SUBAPPLICATION Uebung_003b3_AX (* Funk 16 Tasten auf DataPanel 16 *)
  (* Standard: 61499-2; Description: Copyright (c) 2023 Meisterschulen am Ostbahnhof This program and the accompanying materials are made available under the terms of the Eclipse Public License 2.0 which is available at https://www.eclipse.org/legal/epl-2.0/ SPDX-License-Identifier: EPL-2.0 *)
  (* Version 1.0, 2023-10-23, Franz Höpfinger, Meisterschulen am Ostbahnhof *)
  PACKAGE Uebungen;
  IMPORT DataPanel::io::MI::DQ::DataPanel_MI_DO::DigitalOutput_1A;
  IMPORT DataPanel::io::MI::DQ::DataPanel_MI_DO::DigitalOutput_1B;
  IMPORT DataPanel::io::MI::DQ::DataPanel_MI_DO::DigitalOutput_2A;
  IMPORT DataPanel::io::MI::DQ::DataPanel_MI_DO::DigitalOutput_2B;
  IMPORT DataPanel::io::MI::DQ::DataPanel_MI_DO::DigitalOutput_3A;
  IMPORT DataPanel::io::MI::DQ::DataPanel_MI_DO::DigitalOutput_3B;
  IMPORT DataPanel::io::MI::DQ::DataPanel_MI_DO::DigitalOutput_4A;
  IMPORT DataPanel::io::MI::DQ::DataPanel_MI_DO::DigitalOutput_4B;
  IMPORT DataPanel::io::MI::DQ::DataPanel_MI_DO::DigitalOutput_5A;
  IMPORT DataPanel::io::MI::DQ::DataPanel_MI_DO::DigitalOutput_5B;
  IMPORT DataPanel::io::MI::DQ::DataPanel_MI_DO::DigitalOutput_6A;
  IMPORT DataPanel::io::MI::DQ::DataPanel_MI_DO::DigitalOutput_6B;
  IMPORT DataPanel::io::MI::DQ::DataPanel_MI_DO::DigitalOutput_7A;
  IMPORT DataPanel::io::MI::DQ::DataPanel_MI_DO::DigitalOutput_7B;
  IMPORT DataPanel::io::MI::DQ::DataPanel_MI_DO::DigitalOutput_8A;
  IMPORT DataPanel::io::MI::const::MI::MI_00;
  IMPORT Funk::io::DI::Funk_DI::DigitalInput_Key_01;
  IMPORT Funk::io::DI::Funk_DI::DigitalInput_Key_02;
  IMPORT Funk::io::DI::Funk_DI::DigitalInput_Key_03;
  IMPORT Funk::io::DI::Funk_DI::DigitalInput_Key_04;
  IMPORT Funk::io::DI::Funk_DI::DigitalInput_Key_05;
  IMPORT Funk::io::DI::Funk_DI::DigitalInput_Key_06;
  IMPORT Funk::io::DI::Funk_DI::DigitalInput_Key_07;
  IMPORT Funk::io::DI::Funk_DI::DigitalInput_Key_08;
  IMPORT Funk::io::DI::Funk_DI::DigitalInput_Key_09;
  IMPORT Funk::io::DI::Funk_DI::DigitalInput_Key_10;
  IMPORT Funk::io::DI::Funk_DI::DigitalInput_Key_11;
  IMPORT Funk::io::DI::Funk_DI::DigitalInput_Key_12;
  IMPORT Funk::io::DI::Funk_DI::DigitalInput_Key_13;
  IMPORT Funk::io::DI::Funk_DI::DigitalInput_Key_14;
  IMPORT Funk::io::DI::Funk_DI::DigitalInput_Key_15;
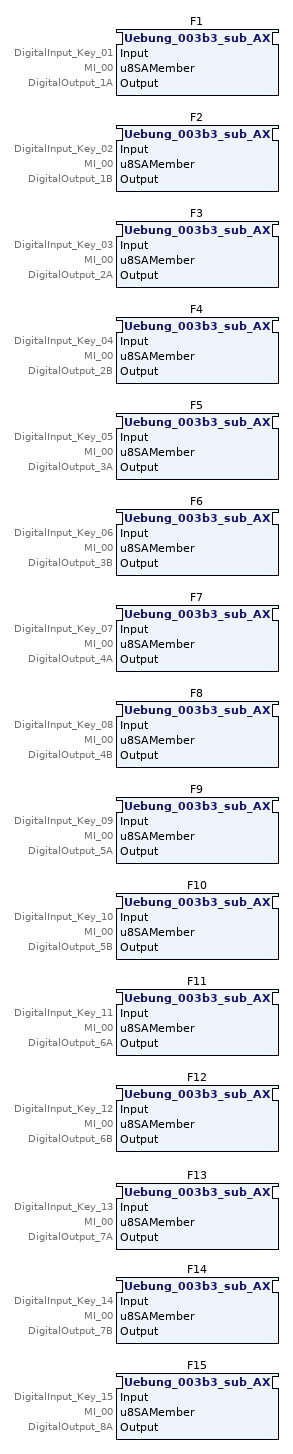
  SUBAPPS
    F1 : Uebungen::Uebung_003b3_sub_AX(Input := DigitalInput_Key_01, u8SAMember := MI_00, Output := DigitalOutput_1A);
    F2 : Uebungen::Uebung_003b3_sub_AX(Input := DigitalInput_Key_02, u8SAMember := MI_00, Output := DigitalOutput_1B);
    F3 : Uebungen::Uebung_003b3_sub_AX(Input := DigitalInput_Key_03, u8SAMember := MI_00, Output := DigitalOutput_2A);
    F4 : Uebungen::Uebung_003b3_sub_AX(Input := DigitalInput_Key_04, u8SAMember := MI_00, Output := DigitalOutput_2B);
    F5 : Uebungen::Uebung_003b3_sub_AX(Input := DigitalInput_Key_05, u8SAMember := MI_00, Output := DigitalOutput_3A);
    F6 : Uebungen::Uebung_003b3_sub_AX(Input := DigitalInput_Key_06, u8SAMember := MI_00, Output := DigitalOutput_3B);
    F7 : Uebungen::Uebung_003b3_sub_AX(Input := DigitalInput_Key_07, u8SAMember := MI_00, Output := DigitalOutput_4A);
    F8 : Uebungen::Uebung_003b3_sub_AX(Input := DigitalInput_Key_08, u8SAMember := MI_00, Output := DigitalOutput_4B);
    F9 : Uebungen::Uebung_003b3_sub_AX(Input := DigitalInput_Key_09, u8SAMember := MI_00, Output := DigitalOutput_5A);
    F10 : Uebungen::Uebung_003b3_sub_AX(Input := DigitalInput_Key_10, u8SAMember := MI_00, Output := DigitalOutput_5B);
    F11 : Uebungen::Uebung_003b3_sub_AX(Input := DigitalInput_Key_11, u8SAMember := MI_00, Output := DigitalOutput_6A);
    F12 : Uebungen::Uebung_003b3_sub_AX(Input := DigitalInput_Key_12, u8SAMember := MI_00, Output := DigitalOutput_6B);
    F13 : Uebungen::Uebung_003b3_sub_AX(Input := DigitalInput_Key_13, u8SAMember := MI_00, Output := DigitalOutput_7A);
    F14 : Uebungen::Uebung_003b3_sub_AX(Input := DigitalInput_Key_14, u8SAMember := MI_00, Output := DigitalOutput_7B);
    F15 : Uebungen::Uebung_003b3_sub_AX(Input := DigitalInput_Key_15, u8SAMember := MI_00, Output := DigitalOutput_8A);
  END_SUBAPPS
END_SUBAPPLICATION
